# EPICS autosave request: iocBoot/ioc13Saturn1/auto_settings_med.req
file "simple_mca_settings.req",  P=13Saturn1:med:, M=mca1
file "dxp_settings.req",         P=13Saturn1:med:, R=dxp1
